# EPICS substitutions: app/Db/pulser.substitutions
file pulser.template
{
    pattern
    { DEV,      PORT,       CSCAN,     DSCAN    }
    { $(DEV),   $(PORT),    $(CSCAN),  $(DSCAN) }
}
